Yaskawa INFORM job: X2_55B(90,0).JBI

/JOB
//NAME X2_55B(90,0)
//POS
///NPOS 393,393,393,16,0,0
///TOOL 0
///POSTYPE PULSE
///PULSE
C00000=-3448,-127156,-102318,81,81770,-493
C00001=187716,-47122,-47867,-37786,88484,55314
C00002=176173,-25216,-33637,-36582,85520,51497
C00003=173223,-25051,-31174,-36235,83113,51076
C00004=172044,-24890,-30122,-36101,82155,50902
C00005=170953,-26782,-31445,-35951,81570,50643
C00006=172044,-24890,-30122,-36101,82155,50902
C00007=171259,-26400,-31421,-35983,81846,50679
C00008=171262,-26151,-29582,-36058,81028,50950
C00009=171259,-26400,-31421,-35983,81846,50679
C00010=171893,-25290,-29924,-36099,81825,50948
C00011=170788,-22386,-27864,-35921,81544,50580
C00012=171893,-25290,-29924,-36099,81825,50948
C00013=172537,-26260,-30983,-36182,82222,51086
C00014=175513,-26532,-33522,-36519,84635,51519
C00015=174876,-38063,-42129,-21725,58370,56921
C00016=172531,-34865,-37156,-20849,56441,56328
C00017=171618,-33525,-35111,-20504,55675,56092
C00018=171621,-33203,-33229,-20744,54744,56283
C00019=171618,-33525,-35111,-20504,55675,56092
C00020=171615,-33256,-33452,-20713,54846,56260
C00021=170195,-32274,-32794,-19931,54588,55694
C00022=171615,-33256,-33452,-20713,54846,56260
C00023=172530,-34620,-35517,-21056,55613,56498
C00024=174875,-37883,-40537,-21925,57545,57094
C00025=186870,-60004,-54988,-28171,58925,61935
C00026=184052,-35224,-20919,-38155,78515,57258
C00027=176072,-20078,-10501,-37523,76109,54673
C00028=173128,-19076,-7343,-37486,73683,54259
C00029=172707,-17410,-5140,-37532,73101,54284
C00030=171611,-19099,-6383,-37450,72543,54005
C00031=172241,-18135,-5678,-37497,72864,54164
C00032=172241,-17854,-4882,-37558,72588,54263
C00033=172241,-17393,-3601,-37659,72145,54424
C00034=172241,-17647,-4307,-37604,72388,54337
C00035=171897,-14890,-2250,-37546,72359,54196
C00036=170935,-12392,-350,-37433,72036,53890
C00037=171859,-14793,-2176,-37541,72348,54182
C00038=174039,-17029,-4295,-37702,73418,54750
C00039=175523,-21167,-9806,-37619,75080,54801
C00040=174791,-34642,-26292,-23834,50951,58585
C00041=172449,-30881,-20835,-23045,48973,57976
C00042=171536,-29314,-18585,-22736,48183,57736
C00043=171539,-28594,-16381,-23083,47273,57969
C00044=171536,-29314,-18585,-22736,48183,57736
C00045=171655,-28757,-16693,-23108,47405,57991
C00046=170233,-27816,-16047,-22270,47093,57375
C00047=171655,-28757,-16693,-23108,47405,57991
C00048=172568,-30347,-18967,-23412,48199,58232
C00049=174914,-34163,-24480,-24186,50191,58839
C00050=188358,-57211,-39729,-31447,52501,64607
C00051=183618,-34426,-20428,-38127,78409,57109
C00052=176138,-20120,-10558,-37527,76149,54687
C00053=173193,-19124,-7405,-37490,73722,54273
C00054=172015,-18635,-6071,-37479,72755,54107
C00055=170924,-20442,-7388,-37397,72187,53833
C00056=172015,-18635,-6071,-37479,72755,54107
C00057=165255,-29463,-17241,-28800,66006,52931
C00058=165259,-28700,-15002,-29010,65138,53168
C00059=172949,-18171,-5639,-37573,73137,54379
C00060=171701,-15066,-3330,-37428,72734,53978
C00061=170868,-12892,-1680,-37330,72456,53714
C00062=171575,-14749,-3089,-37415,72693,53939
C00063=173186,-16870,-5921,-37451,73915,54202
C00064=175516,-21166,-9805,-37619,75076,54799
C00065=174830,-34639,-26268,-23859,50951,58604
C00066=172486,-30879,-20811,-23071,48971,57995
C00067=171574,-29313,-18562,-22761,48182,57754
C00068=171578,-28593,-16359,-23108,47271,57989
C00069=171574,-29313,-18562,-22761,48182,57754
C00070=171610,-28709,-16681,-23077,47409,57968
C00071=170190,-27766,-16033,-22239,47097,57353
C00072=171610,-28709,-16681,-23077,47409,57968
C00073=172523,-30299,-18955,-23380,48203,58209
C00074=174867,-34115,-24469,-24155,50194,58817
C00075=185275,-52966,-37377,-29840,52016,63269
C00076=182622,-32832,-19313,-38072,78076,56798
C00077=176255,-20464,-10741,-37545,76148,54738
C00078=173302,-19472,-7592,-37510,73718,54322
C00079=166116,-18702,-10817,-27686,73217,51023
C00080=166116,-18293,-9498,-27768,72681,51157
C00081=166116,-18702,-10817,-27686,73217,51023
C00082=171916,-17477,-4832,-37501,72578,54128
C00083=171280,-18444,-5544,-37452,72254,53965
C00084=171916,-17477,-4832,-37501,72578,54128
C00085=171570,-15823,-3871,-37423,72632,53954
C00086=170693,-13537,-2145,-37315,72345,53674
C00087=172061,-15821,-3938,-37462,72881,54082
C00088=175486,-21192,-9869,-37613,75083,54783
C00089=174896,-34716,-26303,-23899,50954,58635
C00090=172550,-30958,-20849,-23113,48973,58025
C00091=171637,-29393,-18600,-22803,48182,57784
C00092=171641,-28672,-16396,-23150,47273,58018
C00093=171637,-29393,-18600,-22803,48182,57784
C00094=171632,-28792,-16755,-23089,47417,57977
C00095=170210,-27851,-16107,-22251,47105,57361
C00096=171632,-28792,-16755,-23089,47417,57977
C00097=172546,-30383,-19029,-23392,48210,58218
C00098=174891,-34198,-24540,-24167,50201,58827
C00099=185175,-52762,-37248,-29786,52001,63226
C00100=183220,-33604,-19766,-38110,78246,56996
C00101=176225,-20142,-10450,-37544,76124,54733
C00102=173278,-19146,-7297,-37511,73697,54320
C00103=172099,-18657,-5963,-37501,72729,54152
C00104=171010,-20466,-7281,-37420,72160,53880
C00105=172099,-18657,-5963,-37501,72729,54152
C00106=166571,-28152,-16357,-29058,66575,53325
C00107=166571,-27514,-14492,-29226,65852,53522
C00108=172387,-18207,-5273,-37561,72696,54290
C00109=171548,-16114,-3724,-37463,72430,54020
C00110=170494,-13362,-1647,-37333,72085,53683
C00111=171073,-14893,-2806,-37405,72277,53868
C00112=172620,-14502,-2513,-37545,72964,54297
C00113=175521,-21123,-9840,-37613,75114,54788
C00114=174873,-34635,-26256,-23884,50959,58623
C00115=172529,-30877,-20800,-23097,48977,58014
C00116=171616,-29311,-18550,-22787,48188,57773
C00117=171620,-28590,-16346,-23134,47277,58007
C00118=171616,-29311,-18550,-22787,48188,57773
C00119=171603,-28722,-16701,-23071,47412,57965
C00120=170183,-27779,-16052,-22233,47100,57348
C00121=171603,-28722,-16701,-23071,47412,57965
C00122=172516,-30312,-18976,-23374,48206,58204
C00123=174861,-34128,-24489,-24150,50197,58813
C00124=179101,-45900,-49438,-15006,88631,21048
C00125=172513,-11584,-31608,-27149,87845,-38123
C00126=172121,-24857,-19443,-68057,77460,-42755
C00127=169629,-22717,-14919,-68300,75121,-42365
C00128=168643,-21776,-13037,-68423,74194,-42203
C00129=168645,-21257,-11383,-68611,73902,-41872
C00130=168643,-21776,-13037,-68423,74194,-42203
C00131=168660,-21339,-11618,-68585,73953,-41915
C00132=167619,-20808,-11231,-68547,73267,-42073
C00133=168660,-21339,-11618,-68585,73953,-41915
C00134=169647,-22299,-13520,-68449,74880,-42078
C00135=172140,-24494,-18094,-68180,77218,-42473
C00136=179100,-27267,-21132,-68321,82065,-41721
C00137=177058,-25517,-19916,-68254,80754,-42063
C00138=172070,-24843,-19439,-68055,77427,-42764
C00139=169578,-22699,-14913,-68297,75090,-42374
C00140=168592,-21759,-13031,-68421,74162,-42212
C00141=168594,-21241,-11375,-68608,73870,-41880
C00142=168592,-21759,-13031,-68421,74162,-42212
C00143=168700,-21363,-11631,-68587,73978,-41908
C00144=167658,-20834,-11246,-68549,73291,-42065
C00145=168700,-21363,-11631,-68587,73978,-41908
C00146=169687,-22325,-13534,-68451,74905,-42070
C00147=172181,-24516,-18104,-68183,77243,-42465
C00148=177058,-25517,-19916,-68254,80754,-42063
C00149=178325,-24532,-19230,-68277,81638,-41928
C00150=172107,-24845,-19446,-68056,77454,-42760
C00151=169616,-22704,-14920,-68297,75115,-42370
C00152=168630,-22174,-14386,-68271,74432,-42481
C00153=168630,-21922,-13548,-68363,74279,-42313
C00154=168630,-22174,-14386,-68271,74432,-42481
C00155=167254,-20761,-13369,-68184,73550,-42717
C00156=168630,-22174,-14386,-68271,74432,-42481
C00157=169618,-22273,-13490,-68449,74858,-42080
C00158=172110,-24469,-18066,-68180,77195,-42476
C00159=178325,-24532,-19230,-68277,81638,-41928
C00160=176815,-23437,-18422,-68227,80649,-42160
C00161=172146,-24955,-19493,-68063,77470,-42744
C00162=169652,-22814,-14970,-68305,75130,-42353
C00163=168665,-21875,-13087,-68429,74203,-42192
C00164=168667,-21355,-11432,-68616,73909,-41860
C00165=168665,-21875,-13087,-68429,74203,-42192
C00166=168662,-21419,-11696,-68583,73957,-41918
C00167=167620,-20888,-11311,-68545,73271,-42076
C00168=168662,-21419,-11696,-68583,73957,-41918
C00169=169650,-22379,-13598,-68447,74884,-42081
C00170=172143,-24573,-18170,-68179,77222,-42475
C00171=176815,-23437,-18422,-68227,80649,-42160
C00172=177723,-27338,-20753,-73480,80899,-41496
C00173=173318,-27034,-20539,-73385,77850,-41980
C00174=170566,-24945,-16343,-73635,75471,-41597
C00175=168745,-21940,-12752,-73770,74001,-41488
C00176=168745,-21543,-11513,-73914,73830,-41233
C00177=168745,-21940,-12752,-73770,74001,-41488
C00178=167687,-21056,-12116,-73735,73288,-41631
C00179=168745,-21940,-12752,-73770,74001,-41488
C00180=170579,-24581,-15077,-73772,75297,-41328
C00181=173331,-26714,-19314,-73495,77675,-41714
C00182=177723,-27338,-20753,-73480,80899,-41496
C00183=178463,-3707,1935,-68390,87302,-39636
C00184=172445,-1687,3602,-68547,83267,-40440
C00185=171155,2365,8138,-68637,82124,-40308
C00186=169346,2928,9772,-68759,80632,-40240
C00187=168978,-317,7268,-68782,80335,-40236
C00188=168639,-4450,3875,-68796,80092,-40264
C00189=168178,-8509,681,-68823,79735,-40271
C00190=167808,-11173,-1351,-68851,79442,-40266
C00191=167512,-13424,-3126,-68866,79215,-40276
C00192=170518,-14544,-5815,-68770,81540,-41125
C00193=171276,-16033,-7526,-68427,80959,-50953
C00194=176138,-7665,-1065,-68313,84347,-50442
C00195=175728,4349,8139,-68463,85593,-40138
C00196=172451,-1962,2819,-68519,83404,-40586
C00197=170217,-243,7278,-68749,81179,-40082
C00198=168682,3850,12028,-68899,79836,-39929
C00199=168320,-294,8663,-68919,79564,-39952
C00200=167945,-5454,4438,-68970,78444,-40143
C00201=167170,-12539,-831,-69280,75932,-44117
C00202=166914,-13716,-1698,-69168,76543,-48053
C00203=168751,-15418,-4687,-68668,78708,-50672
C00204=171281,-16312,-8291,-68386,81093,-51093
C00205=176223,-7788,-1720,-68290,84540,-50575
C00206=175841,4947,9210,-68476,85532,-39971
C00207=172439,-1632,3648,-68547,83263,-40441
C00208=170207,122,8144,-68792,81039,-39934
C00209=169582,3762,12383,-68907,80337,-39699
C00210=169205,-1273,8190,-68921,80079,-39742
C00211=168949,-4829,5248,-68968,79052,-39936
C00212=168747,-7437,3182,-69019,78039,-40097
C00213=168400,-11411,49,-69099,75859,-40464
C00214=168049,-14366,-2154,-69161,74008,-40742
C00215=167878,-15531,-2988,-69182,74134,-40673
C00216=167909,-10329,250,-68068,79474,-40087
C00217=167962,-8065,2008,-67933,82039,-39608
C00218=168741,-15055,-3851,-68723,78573,-50532
C00219=171270,-15979,-7485,-68426,80956,-50955
C00220=176912,-6106,181,-68292,84880,-50353
C00221=175080,3284,7783,-68495,85030,-40084
C00222=172448,-1714,3579,-68547,83270,-40439
C00223=170215,38,8073,-68791,81044,-39933
C00224=169530,3059,11777,-68909,80304,-39708
C00225=169167,-1208,8273,-68926,80049,-39741
C00226=168895,-5244,4985,-68982,78994,-39919
C00227=168721,-7713,2972,-69022,78019,-40095
C00228=168321,-11533,70,-69119,75776,-40439
C00229=168019,-14335,-2124,-69163,73986,-40743
C00230=167869,-15557,-2996,-69185,74125,-40670
C00231=167778,-15678,-3083,-69135,76109,-40273
C00232=168308,-1085,8366,-68428,86286,-38506
C00233=168749,-15137,-3913,-68724,78577,-50529
C00234=171279,-16061,-7546,-68427,80961,-50952
C00235=176975,-6087,196,-68290,84923,-50345
C00236=175436,4075,8459,-68486,85264,-40032
C00237=172442,-1659,3624,-68547,83265,-40441
C00238=170209,94,8121,-68791,81041,-39934
C00239=169521,3688,12369,-68916,80282,-39689
C00240=169178,-1205,8258,-68923,80058,-39744
C00241=168951,-4837,5280,-68974,79043,-39923
C00242=168871,-5612,4655,-68979,78986,-39928
C00243=168324,-12009,-390,-69107,75794,-40458
C00244=167899,-15618,-3071,-69178,74154,-40675
C00245=168117,-12377,-741,-68965,78498,-39952
C00246=168316,-5643,4501,-68586,83486,-39095
C00247=169562,-13065,-2936,-68632,79303,-50620
C00248=171273,-16006,-7506,-68427,80957,-50954
C00249=176232,-7453,-896,-68311,84412,-50431
C00250=176110,15147,-7571,-16904,97824,-889
C00251=169929,-46392,-55011,-1489,81060,44357
C00252=178847,-41200,-24878,-45467,45731,82659
C00253=176214,-37608,-19575,-45318,43383,82417
C00254=175671,-33630,-15830,-45260,42922,82348
C00255=175825,-32530,-15066,-45264,43068,82357
C00256=178049,-27664,-11799,-47846,47063,84437
C00257=178346,-25405,-10245,-47840,47361,84442
C00258=178686,-23359,-8771,-47863,47635,84481
C00259=179298,-27755,-13076,-47829,48231,84493
C00260=181844,-30788,-18177,-47745,50662,84564
C00261=174365,-16035,-7463,-23225,65722,49139
C00262=172039,-13164,-2259,-22946,63476,48682
C00263=170681,-8939,2085,-22689,62636,48310
C00264=168716,-14063,-1663,-20852,60530,45982
C00265=168210,-15866,-3076,-20705,60349,45807
C00266=167705,-17394,-4214,-20570,60144,45641
C00267=168908,-9574,565,-22819,69097,42788
C00268=170886,-12368,-2848,-23069,70258,43317
C00269=173248,-14965,-7813,-23249,72509,43767
C00270=172938,-13150,-5784,-34661,81894,69122
C00271=170592,-13671,-3251,-34736,79423,68935
C00272=169013,-12050,-743,-34751,78192,68673
C00273=168391,-10413,528,-34716,77985,68483
C00274=167212,-7347,2971,-34654,77563,68126
C00275=167368,-11109,1537,-37136,72671,67957
C00276=169061,-13362,-1350,-37170,73898,68258
C00277=171567,-13522,-4340,-37101,76395,68464
C00278=179365,-30795,-16721,-37645,78767,70970
C00279=189901,-62154,-47134,-47848,53538,74187
C00280=178827,-45311,-37716,-41873,49979,80234
C00281=176196,-42115,-32789,-41416,47672,79900
C00282=175621,-38539,-29280,-41324,47154,79828
C00283=175830,-37491,-28575,-41455,47414,79922
C00284=176568,-36338,-27837,-42536,48701,80694
C00285=177913,-33249,-25871,-44214,51091,81919
C00286=178266,-30726,-24137,-44250,51432,81940
C00287=178622,-27514,-21859,-44263,51790,81950
C00288=179281,-31896,-26227,-44296,52442,81981
C00289=181826,-34468,-30902,-44523,54848,82142
C00290=174316,-20812,-35323,-21564,79352,46486
C00291=171992,-19198,-31213,-21065,77169,46035
C00292=171153,-17227,-28586,-20882,76391,45864
C00293=169593,-21753,-31892,-19124,74559,43851
C00294=168812,-24435,-33772,-18910,74171,43627
C00295=168062,-26842,-35420,-18710,73789,43414
C00296=169770,-16807,-29422,-21714,83022,40480
C00297=169547,-17498,-29909,-21673,82913,40417
C00298=170841,-17822,-31354,-21899,83925,40699
C00299=173201,-19163,-35240,-22305,86132,41137
C00300=172907,-17608,-30546,-34532,92651,65775
C00301=170563,-19319,-28972,-34275,90177,65595
C00302=169577,-19876,-27906,-34181,88999,65557
C00303=168529,-16782,-25766,-34081,88801,65197
C00304=167923,-15565,-24727,-34164,88196,64970
C00305=167964,-19498,-26291,-35768,83354,64607
C00306=169032,-19661,-27621,-35877,84402,64708
C00307=171538,-18685,-29668,-36163,86886,64924
C00308=178275,-34785,-40895,-36932,88626,67129
C00309=191077,-58387,-34695,-51576,50395,82052
C00310=178834,-41148,-24847,-45459,45731,82652
C00311=176205,-37556,-19542,-45310,43382,82411
C00312=175763,-33644,-15876,-45294,42982,82374
C00313=178032,-28543,-12452,-47893,47019,84460
C00314=178404,-25994,-10760,-47830,47404,84453
C00315=178792,-23615,-9141,-47838,47760,84471
C00316=179288,-27703,-13041,-47822,48229,84487
C00317=181832,-30737,-18143,-47737,50660,84558
C00318=174357,-15982,-7423,-23222,65723,49136
C00319=172031,-13111,-2218,-22944,63477,48679
C00320=170520,-8947,1823,-22613,62739,48224
C00321=170034,-11263,-69,-22486,62583,48061
C00322=169470,-13204,-1541,-22355,62344,47883
C00323=168361,-16702,-4145,-22089,61865,47531
C00324=168865,-9474,239,-22775,69314,42731
C00325=170879,-12314,-2806,-23068,70257,43314
C00326=173241,-14911,-7773,-23247,72510,43764
C00327=172940,-13092,-5769,-34660,81912,69117
C00328=170596,-13616,-3238,-34734,79442,68930
C00329=168939,-11997,-1091,-34723,78363,68588
C00330=168389,-10110,342,-34686,78206,68407
C00331=167070,-6484,3213,-34619,77749,68010
C00332=167299,-10933,1331,-37095,72823,67875
C00333=169065,-13308,-1339,-37166,73916,68253
C00334=171571,-13466,-4327,-37098,76413,68459
C00335=178312,-28732,-15356,-37588,78485,70620
C00336=191277,-58648,-34832,-51660,50475,82922
C00337=178852,-41226,-24894,-45472,45733,82663
C00338=176220,-37634,-19591,-45323,43383,82420
C00339=175685,-33946,-16007,-45315,42889,82377
C00340=175835,-32522,-15044,-45277,43065,82364
C00341=178144,-27733,-11903,-47880,47136,84457
C00342=178393,-25451,-10265,-47844,47377,84457
C00343=178672,-23784,-9159,-47826,47648,84464
C00344=179304,-27780,-13094,-47832,48232,84495
C00345=181850,-30813,-18194,-47748,50663,84567
C00346=174368,-16065,-7493,-23225,65726,49140
C00347=172043,-13195,-2289,-22946,63480,48682
C00348=171164,-7550,3016,-22790,62898,48455
C00349=170866,-8989,1826,-22712,62814,48348
C00350=170143,-11437,8,-22546,62486,48122
C00351=169193,-14739,-2522,-22318,62099,47819
C00352=169244,-9393,584,-22743,68342,43554
C00353=170889,-12399,-2879,-23069,70262,43318
C00354=173252,-14995,-7844,-23249,72513,43768
C00355=172951,-13173,-5831,-34660,81913,69121
C00356=170605,-13697,-3300,-34735,79444,68934
C00357=169521,-10404,420,-34756,78511,68787
C00358=168984,-8925,1564,-34730,78334,68616
C00359=167678,-5351,4395,-34667,77878,68219
C00360=170004,-9650,4792,-41331,72244,71659
C00361=169881,-12181,-477,-37221,74307,68468
C00362=171580,-13547,-4389,-37099,76414,68462
C00363=179014,-30130,-16303,-37625,78683,70850
C00364=192370,-59799,-35433,-52082,50945,77766
C00365=178840,-41174,-24863,-45463,45731,82656
C00366=176209,-37582,-19559,-45314,43383,82414
C00367=175858,-33709,-16041,-45280,43083,82373
C00368=175847,-33097,-15509,-45291,43063,82377
C00369=178181,-27613,-11893,-47837,47190,84441
C00370=178483,-25011,-10021,-47840,47478,84452
C00371=178690,-24031,-9393,-47845,47668,84462
C00372=179293,-27729,-13059,-47826,48231,84490
C00373=181839,-30763,-18160,-47741,50661,84561
C00374=174361,-16008,-7442,-23223,65722,49137
C00375=172034,-13138,-2238,-22945,63477,48680
C00376=171207,-7845,2636,-22781,62991,48446
C00377=170272,-11167,86,-22561,62606,48149
C00378=169822,-12966,-1346,-22450,62442,48001
C00379=168964,-15587,-3284,-22246,62068,47732
C00380=173943,-1511,8904,-29878,72865,47458
C00381=172046,-12965,-4840,-23146,71432,43525
C00382=173245,-14938,-7793,-23248,72510,43766
C00383=172944,-13119,-5789,-34660,81912,69118
C00384=170599,-13643,-3259,-34734,79442,68931
C00385=169526,-10552,102,-34744,78615,68757
C00386=169161,-9437,984,-34729,78491,68643
C00387=167403,-4604,4769,-34640,77906,68103
C00388=171806,-13548,4066,-45686,69255,74076
C00389=169068,-13335,-1360,-37167,73916,68254
C00390=171574,-13493,-4347,-37099,76413,68460
C00391=179991,-31915,-17499,-37671,78963,71169
C00392=-3448,-127156,-102318,81,81770,-493
BC00000=88064,523889,1075193
BC00001=92522,523889,1075139
BC00002=92522,523889,1075139
BC00003=92522,523889,1075139
BC00004=92522,523889,1075139
BC00005=92522,523889,1075139
BC00006=92522,523889,1075139
BC00007=92522,523889,1075139
BC00008=92522,523889,1075139
BC00009=92522,523889,1075139
BC00010=92522,523889,1075139
BC00011=92522,523889,1075139
BC00012=92522,523889,1075139
BC00013=92522,523889,1075139
BC00014=92522,523889,1075139
BC00015=117731,523889,1075139
BC00016=117731,523889,1075139
BC00017=117731,523889,1075139
BC00018=117731,523889,1075139
BC00019=117731,523889,1075139
BC00020=117731,523889,1075139
BC00021=117731,523889,1075139
BC00022=117731,523889,1075139
BC00023=117731,523889,1075139
BC00024=117731,523889,1075139
BC00025=117731,523889,1075139
BC00026=92535,523889,1039496
BC00027=92535,523889,1039496
BC00028=92535,523889,1039496
BC00029=92535,523889,1039496
BC00030=92535,523889,1039496
BC00031=92535,523889,1039496
BC00032=92535,523889,1039496
BC00033=92535,523889,1039496
BC00034=92535,523889,1039496
BC00035=92535,523889,1039496
BC00036=92535,523889,1039496
BC00037=92535,523889,1039496
BC00038=92535,523889,1039496
BC00039=92535,523889,1039496
BC00040=117708,523889,1001261
BC00041=117708,523889,1001261
BC00042=117708,523889,1001261
BC00043=117708,523889,1001261
BC00044=117708,523889,1001261
BC00045=117708,523889,1001261
BC00046=117708,523889,1001261
BC00047=117708,523889,1001261
BC00048=117708,523889,1001261
BC00049=117708,523889,1001261
BC00050=117708,523889,1001261
BC00051=92605,523889,877547
BC00052=92605,523889,877547
BC00053=92605,523889,877547
BC00054=92605,523889,877547
BC00055=92605,523889,877547
BC00056=92605,523889,877547
BC00057=92605,523889,877547
BC00058=92605,523889,877547
BC00059=92605,523889,877547
BC00060=92605,523889,877547
BC00061=92605,523889,877547
BC00062=92605,523889,877547
BC00063=92605,523889,877547
BC00064=92605,523889,877547
BC00065=117541,523889,839285
BC00066=117541,523889,839285
BC00067=117541,523889,839285
BC00068=117541,523889,839285
BC00069=117541,523889,839285
BC00070=117541,523889,839285
BC00071=117541,523889,839285
BC00072=117541,523889,839285
BC00073=117541,523889,839285
BC00074=117541,523889,839285
BC00075=117541,523889,839285
BC00076=92484,523889,715304
BC00077=92484,523889,715304
BC00078=92484,523889,715304
BC00079=92484,523889,715304
BC00080=92484,523889,715304
BC00081=92484,523889,715304
BC00082=92484,523889,715304
BC00083=92484,523889,715304
BC00084=92484,523889,715304
BC00085=92484,523889,715304
BC00086=92484,523889,715304
BC00087=92484,523889,715304
BC00088=92484,523889,715304
BC00089=117712,523889,677277
BC00090=117712,523889,677277
BC00091=117712,523889,677277
BC00092=117712,523889,677277
BC00093=117712,523889,677277
BC00094=117712,523889,677277
BC00095=117712,523889,677277
BC00096=117712,523889,677277
BC00097=117712,523889,677277
BC00098=117712,523889,677277
BC00099=117712,523889,677277
BC00100=92665,523889,553782
BC00101=92665,523889,553782
BC00102=92665,523889,553782
BC00103=92665,523889,553782
BC00104=92665,523889,553782
BC00105=92665,523889,553782
BC00106=92665,523889,553782
BC00107=92665,523889,553782
BC00108=92665,523889,553782
BC00109=92665,523889,553782
BC00110=92665,523889,553782
BC00111=92665,523889,553782
BC00112=92665,523889,553782
BC00113=92665,523889,553782
BC00114=117593,523889,515943
BC00115=117593,523889,515943
BC00116=117593,523889,515943
BC00117=117593,523889,515943
BC00118=117593,523889,515943
BC00119=117593,523889,515943
BC00120=117593,523889,515943
BC00121=117593,523889,515943
BC00122=117593,523889,515943
BC00123=117593,523889,515943
BC00124=88297,523889,479689
BC00125=36680,523889,415813
BC00126=28310,523889,405455
BC00127=28310,523889,405455
BC00128=29106,522353,405455
BC00129=29106,522353,405455
BC00130=29106,522353,405455
BC00131=29106,522353,405455
BC00132=29106,522353,405455
BC00133=29106,522353,405455
BC00134=29106,522353,405455
BC00135=29106,522353,405455
BC00136=29106,522353,405455
BC00137=29225,522353,566726
BC00138=29225,522353,566726
BC00139=29225,522353,566726
BC00140=29225,522353,566726
BC00141=29225,522353,566726
BC00142=29225,522353,566726
BC00143=29225,522353,566726
BC00144=29225,522353,566726
BC00145=29225,522353,566726
BC00146=29225,522353,566726
BC00147=29225,522353,566726
BC00148=29225,522353,566726
BC00149=28944,522353,728798
BC00150=28944,522353,728798
BC00151=28944,522353,728798
BC00152=28944,522353,728798
BC00153=28944,522353,728798
BC00154=28944,522353,728798
BC00155=28944,522353,728798
BC00156=28944,522353,728798
BC00157=28944,522353,728798
BC00158=28944,522353,728798
BC00159=28944,522353,728798
BC00160=29066,522353,891103
BC00161=29066,522353,891103
BC00162=29066,522353,891103
BC00163=29066,522353,891103
BC00164=29066,522353,891103
BC00165=29066,522353,891103
BC00166=29066,522353,891103
BC00167=29066,522353,891103
BC00168=29066,522353,891103
BC00169=29066,522353,891103
BC00170=29066,522353,891103
BC00171=29066,522353,891103
BC00172=26330,522353,1022235
BC00173=26330,522353,1022235
BC00174=26330,522353,1022235
BC00175=26330,522353,1022235
BC00176=26330,522353,1022235
BC00177=26330,522353,1022235
BC00178=26330,522353,1022235
BC00179=26330,522353,1022235
BC00180=26330,522353,1022235
BC00181=26330,522353,1022235
BC00182=26330,522353,1022235
BC00183=28832,522353,754426
BC00184=28036,523889,754426
BC00185=28036,523889,754426
BC00186=28832,522353,754426
BC00187=28832,522353,754426
BC00188=28832,522353,754426
BC00189=28832,522353,754426
BC00190=28832,522353,754426
BC00191=28832,522353,754426
BC00192=28832,522353,754426
BC00193=28832,522353,754426
BC00194=28832,522353,754426
BC00195=28825,522353,1075139
BC00196=28825,522353,1075139
BC00197=28825,522353,1075139
BC00198=28825,522353,1075139
BC00199=28825,522353,1075139
BC00200=28825,522353,1075139
BC00201=28825,522353,1075139
BC00202=28825,522353,1075139
BC00203=28825,522353,1075139
BC00204=28825,522353,1075139
BC00205=28825,522353,1075139
BC00206=28839,522353,431016
BC00207=28839,522353,431016
BC00208=28839,522353,431016
BC00209=28839,522353,431016
BC00210=28839,522353,431016
BC00211=28839,522353,431016
BC00212=28839,522353,431016
BC00213=28839,522353,431016
BC00214=28839,522353,431016
BC00215=28839,522353,431016
BC00216=28839,522353,431016
BC00217=28839,522353,431016
BC00218=28839,522353,431016
BC00219=28839,522353,431016
BC00220=28839,522353,431016
BC00221=28829,522353,916535
BC00222=28829,522353,916535
BC00223=28829,522353,916535
BC00224=28829,522353,916535
BC00225=28829,522353,916535
BC00226=28829,522353,916535
BC00227=28829,522353,916535
BC00228=28829,522353,916535
BC00229=28829,522353,916535
BC00230=28829,522353,916535
BC00231=28829,522353,916535
BC00232=28829,522353,916535
BC00233=28829,522353,916535
BC00234=28829,522353,916535
BC00235=28829,522353,916535
BC00236=28835,522353,592318
BC00237=28835,522353,592318
BC00238=28835,522353,592318
BC00239=28835,522353,592318
BC00240=28835,522353,592318
BC00241=28835,522353,592318
BC00242=28835,522353,592318
BC00243=28835,522353,592318
BC00244=28835,522353,592318
BC00245=28835,522352,592316
BC00246=28835,522352,592316
BC00247=28835,522353,592318
BC00248=28835,522353,592318
BC00249=28835,522353,592318
BC00250=67844,522353,695135
BC00251=94775,523889,768216
BC00252=112941,523889,816097
BC00253=112941,523889,816097
BC00254=112941,523889,816097
BC00255=112941,523889,816097
BC00256=112941,523889,816097
BC00257=112941,523889,816097
BC00258=112941,523889,816097
BC00259=112941,523889,816097
BC00260=112941,523889,816097
BC00261=118115,523889,907170
BC00262=118115,523889,907170
BC00263=118115,523889,907170
BC00264=118115,523889,907170
BC00265=118115,523889,907170
BC00266=118115,523889,907170
BC00267=118115,523889,907170
BC00268=118115,523889,907170
BC00269=118115,523889,907170
BC00270=88032,523889,888291
BC00271=88032,523889,888291
BC00272=88032,523889,888291
BC00273=88032,523889,888291
BC00274=88032,523889,888291
BC00275=88032,523889,888291
BC00276=88032,523889,888291
BC00277=88032,523889,888291
BC00278=88032,523889,888291
BC00279=112934,523889,1075139
BC00280=112934,523889,1075139
BC00281=112934,523889,1075139
BC00282=112934,523889,1075139
BC00283=112934,523889,1075139
BC00284=112934,523889,1075139
BC00285=112934,523889,1075139
BC00286=112934,523889,1075139
BC00287=112934,523889,1075139
BC00288=112934,523889,1075139
BC00289=112934,523889,1075139
BC00290=118108,523889,1075139
BC00291=118108,523889,1075139
BC00292=118108,523889,1075139
BC00293=118108,523889,1075139
BC00294=118108,523889,1075139
BC00295=118108,523889,1075139
BC00296=118108,523889,1075139
BC00297=118108,523889,1075139
BC00298=118108,523889,1075139
BC00299=118108,523889,1075139
BC00300=88054,523889,1075139
BC00301=88054,523889,1075139
BC00302=88054,523888,1075137
BC00303=88054,523889,1075139
BC00304=88054,523889,1075139
BC00305=88054,523889,1075139
BC00306=88054,523889,1075139
BC00307=88054,523889,1075139
BC00308=88054,523889,1075139
BC00309=112948,523889,492686
BC00310=112948,523889,492686
BC00311=112948,523889,492686
BC00312=112948,523889,492686
BC00313=112948,523889,492686
BC00314=112948,523889,492686
BC00315=112948,523889,492686
BC00316=112948,523889,492686
BC00317=112948,523889,492686
BC00318=118122,523889,583760
BC00319=118122,523889,583760
BC00320=118122,523889,583760
BC00321=118122,523889,583760
BC00322=118122,523889,583760
BC00323=118122,523889,583760
BC00324=118122,523889,583760
BC00325=118122,523889,583760
BC00326=118122,523889,583760
BC00327=88067,523889,564693
BC00328=88067,523889,564693
BC00329=88067,523889,564693
BC00330=88067,523889,564693
BC00331=88067,523889,564693
BC00332=88067,523889,564693
BC00333=88067,523889,564693
BC00334=88067,523889,564693
BC00335=88067,523889,564693
BC00336=112938,523889,978206
BC00337=112938,523889,978206
BC00338=112938,523889,978206
BC00339=112938,523889,978206
BC00340=112938,523889,978206
BC00341=112938,523889,978206
BC00342=112938,523889,978206
BC00343=112938,523889,978206
BC00344=112938,523889,978206
BC00345=112938,523889,978206
BC00346=118112,523889,1069230
BC00347=118112,523889,1069230
BC00348=118112,523889,1069230
BC00349=118112,523889,1069230
BC00350=118112,523889,1069230
BC00351=118112,523889,1069230
BC00352=118111,523889,1069227
BC00353=118112,523889,1069230
BC00354=118112,523889,1069230
BC00355=88057,523889,1050213
BC00356=88057,523889,1050213
BC00357=88057,523889,1050213
BC00358=88057,523889,1050213
BC00359=88057,523889,1050213
BC00360=88057,523889,1050213
BC00361=88057,523889,1050213
BC00362=88057,523889,1050213
BC00363=88057,523889,1050213
BC00364=112944,523889,653988
BC00365=112944,523889,653988
BC00366=112944,523889,653988
BC00367=112944,523889,653988
BC00368=112944,523889,653988
BC00369=112944,523889,653988
BC00370=112944,523889,653988
BC00371=112944,523889,653988
BC00372=112944,523889,653988
BC00373=112944,523889,653988
BC00374=118118,523889,745062
BC00375=118118,523889,745062
BC00376=118118,523889,745062
BC00377=118118,523889,745062
BC00378=118118,523889,745062
BC00379=118118,523889,745062
BC00380=118118,523889,745062
BC00381=118118,523889,745062
BC00382=118118,523889,745062
BC00383=88064,523889,725995
BC00384=88064,523889,725995
BC00385=88064,523889,725995
BC00386=88064,523889,725995
BC00387=88064,523889,725995
BC00388=88064,523889,725995
BC00389=88064,523889,725995
BC00390=88064,523889,725995
BC00391=88064,555625,725995
BC00392=88064,523889,1075193
EC00000=-798156,-183832
EC00001=-798156,-183832
EC00002=-798156,-183832
EC00003=-798156,-183832
EC00004=-798156,-183832
EC00005=-798156,-183832
EC00006=-798156,-183832
EC00007=-798156,-183832
EC00008=-798156,-183832
EC00009=-798156,-183832
EC00010=-798156,-183832
EC00011=-798156,-183832
EC00012=-798156,-183832
EC00013=-798156,-183832
EC00014=-798156,-183832
EC00015=-798156,-183832
EC00016=-798156,-183832
EC00017=-798156,-183832
EC00018=-798156,-183832
EC00019=-798156,-183832
EC00020=-798156,-183832
EC00021=-798156,-183832
EC00022=-798156,-183832
EC00023=-798156,-183832
EC00024=-798156,-183832
EC00025=-798156,-183832
EC00026=-798156,-183832
EC00027=-798156,-183832
EC00028=-798156,-183832
EC00029=-798156,-183832
EC00030=-798156,-183832
EC00031=-798156,-183832
EC00032=-798156,-183832
EC00033=-798156,-183832
EC00034=-798156,-183832
EC00035=-798156,-183832
EC00036=-798156,-183832
EC00037=-798156,-183832
EC00038=-798156,-183832
EC00039=-798156,-183832
EC00040=-798156,-183832
EC00041=-798156,-183832
EC00042=-798156,-183832
EC00043=-798156,-183832
EC00044=-798156,-183832
EC00045=-798156,-183832
EC00046=-798156,-183832
EC00047=-798156,-183832
EC00048=-798156,-183832
EC00049=-798156,-183832
EC00050=-798156,-183832
EC00051=-798156,-183832
EC00052=-798156,-183832
EC00053=-798156,-183832
EC00054=-798156,-183832
EC00055=-798156,-183832
EC00056=-798156,-183832
EC00057=-798156,-183832
EC00058=-798156,-183832
EC00059=-798156,-183832
EC00060=-798156,-183832
EC00061=-798156,-183832
EC00062=-798156,-183832
EC00063=-798156,-183832
EC00064=-798156,-183832
EC00065=-798156,-183832
EC00066=-798156,-183832
EC00067=-798156,-183832
EC00068=-798156,-183832
EC00069=-798156,-183832
EC00070=-798156,-183832
EC00071=-798156,-183832
EC00072=-798156,-183832
EC00073=-798156,-183832
EC00074=-798156,-183832
EC00075=-798156,-183832
EC00076=-798156,-183832
EC00077=-798156,-183832
EC00078=-798156,-183832
EC00079=-798156,-183832
EC00080=-798156,-183832
EC00081=-798156,-183832
EC00082=-798156,-183832
EC00083=-798156,-183832
EC00084=-798156,-183832
EC00085=-798156,-183832
EC00086=-798156,-183832
EC00087=-798156,-183832
EC00088=-798156,-183832
EC00089=-798156,-183832
EC00090=-798156,-183832
EC00091=-798156,-183832
EC00092=-798156,-183832
EC00093=-798156,-183832
EC00094=-798156,-183832
EC00095=-798156,-183832
EC00096=-798156,-183832
EC00097=-798156,-183832
EC00098=-798156,-183832
EC00099=-798156,-183832
EC00100=-798156,-183832
EC00101=-798156,-183832
EC00102=-798156,-183832
EC00103=-798156,-183832
EC00104=-798156,-183832
EC00105=-798156,-183832
EC00106=-798156,-183832
EC00107=-798156,-183832
EC00108=-798156,-183832
EC00109=-798156,-183832
EC00110=-798156,-183832
EC00111=-798156,-183832
EC00112=-798156,-183832
EC00113=-798156,-183832
EC00114=-798156,-183832
EC00115=-798156,-183832
EC00116=-798156,-183832
EC00117=-798156,-183832
EC00118=-798156,-183832
EC00119=-798156,-183832
EC00120=-798156,-183832
EC00121=-798156,-183832
EC00122=-798156,-183832
EC00123=-798156,-183832
EC00124=-798156,-183832
EC00125=-798156,-183832
EC00126=-798156,-183832
EC00127=-798156,-183832
EC00128=-798156,-183832
EC00129=-798156,-183832
EC00130=-798156,-183832
EC00131=-798156,-183832
EC00132=-798156,-183832
EC00133=-798156,-183832
EC00134=-798156,-183832
EC00135=-798156,-183832
EC00136=-798156,-183832
EC00137=-798156,-183832
EC00138=-798156,-183832
EC00139=-798156,-183832
EC00140=-798156,-183832
EC00141=-798156,-183832
EC00142=-798156,-183832
EC00143=-798156,-183832
EC00144=-798156,-183832
EC00145=-798156,-183832
EC00146=-798156,-183832
EC00147=-798156,-183832
EC00148=-798156,-183832
EC00149=-798156,-183832
EC00150=-798156,-183832
EC00151=-798156,-183832
EC00152=-798156,-183832
EC00153=-798156,-183832
EC00154=-798156,-183832
EC00155=-798156,-183832
EC00156=-798156,-183832
EC00157=-798156,-183832
EC00158=-798156,-183832
EC00159=-798156,-183832
EC00160=-798156,-183832
EC00161=-798156,-183832
EC00162=-798156,-183832
EC00163=-798156,-183832
EC00164=-798156,-183832
EC00165=-798156,-183832
EC00166=-798156,-183832
EC00167=-798156,-183832
EC00168=-798156,-183832
EC00169=-798156,-183832
EC00170=-798156,-183832
EC00171=-798156,-183832
EC00172=-798156,-183832
EC00173=-798156,-183832
EC00174=-798156,-183832
EC00175=-798156,-183832
EC00176=-798156,-183832
EC00177=-798156,-183832
EC00178=-798156,-183832
EC00179=-798156,-183832
EC00180=-798156,-183832
EC00181=-798156,-183832
EC00182=-798156,-183832
EC00183=-798156,-183832
EC00184=-798156,-183832
EC00185=-798156,-183832
EC00186=-798156,-183832
EC00187=-798156,-183832
EC00188=-798156,-183832
EC00189=-798156,-183832
EC00190=-798156,-183832
EC00191=-798156,-183832
EC00192=-798156,-183832
EC00193=-798156,-183832
EC00194=-798156,-183832
EC00195=-798156,-183832
EC00196=-798156,-183832
EC00197=-798156,-183832
EC00198=-798156,-183832
EC00199=-798156,-183832
EC00200=-798156,-183832
EC00201=-798156,-183832
EC00202=-798156,-183832
EC00203=-798156,-183832
EC00204=-798156,-183832
EC00205=-798156,-183832
EC00206=-798156,-183832
EC00207=-798156,-183832
EC00208=-798156,-183832
EC00209=-798156,-183832
EC00210=-798156,-183832
EC00211=-798156,-183832
EC00212=-798156,-183832
EC00213=-798156,-183832
EC00214=-798156,-183832
EC00215=-798156,-183832
EC00216=-798156,-183832
EC00217=-798156,-183832
EC00218=-798156,-183832
EC00219=-798156,-183832
EC00220=-798156,-183832
EC00221=-798156,-183832
EC00222=-798156,-183832
EC00223=-798156,-183832
EC00224=-798156,-183832
EC00225=-798156,-183832
EC00226=-798156,-183832
EC00227=-798156,-183832
EC00228=-798156,-183832
EC00229=-798156,-183832
EC00230=-798156,-183832
EC00231=-798156,-183832
EC00232=-798156,-183832
EC00233=-798156,-183832
EC00234=-798156,-183832
EC00235=-798156,-183832
EC00236=-798156,-183832
EC00237=-798156,-183832
EC00238=-798156,-183832
EC00239=-798156,-183832
EC00240=-798156,-183832
EC00241=-798156,-183832
EC00242=-798156,-183832
EC00243=-798156,-183832
EC00244=-798156,-183832
EC00245=-798155,-183832
EC00246=-798155,-183832
EC00247=-798156,-183832
EC00248=-798156,-183832
EC00249=-798156,-183832
EC00250=-798156,-183832
EC00251=-798156,-183832
EC00252=-798156,-183832
EC00253=-798156,-183832
EC00254=-798156,-183832
EC00255=-798156,-183832
EC00256=-798156,-183832
EC00257=-798156,-183832
EC00258=-798156,-183832
EC00259=-798156,-183832
EC00260=-798156,-183832
EC00261=-798156,-183832
EC00262=-798156,-183832
EC00263=-798156,-183832
EC00264=-798156,-183832
EC00265=-798156,-183832
EC00266=-798156,-183832
EC00267=-798156,-183832
EC00268=-798156,-183832
EC00269=-798156,-183832
EC00270=-798156,-183832
EC00271=-798156,-183832
EC00272=-798156,-183832
EC00273=-798156,-183832
EC00274=-798156,-183832
EC00275=-798156,-183832
EC00276=-798156,-183832
EC00277=-798156,-183832
EC00278=-798156,-183832
EC00279=-798156,-183832
EC00280=-798156,-183832
EC00281=-798156,-183832
EC00282=-798156,-183832
EC00283=-798156,-183832
EC00284=-798156,-183832
EC00285=-798156,-183832
EC00286=-798156,-183832
EC00287=-798156,-183832
EC00288=-798156,-183832
EC00289=-798156,-183832
EC00290=-798156,-183832
EC00291=-798156,-183832
EC00292=-798156,-183832
EC00293=-798156,-183832
EC00294=-798156,-183832
EC00295=-798156,-183832
EC00296=-798156,-183832
EC00297=-798156,-183832
EC00298=-798156,-183832
EC00299=-798156,-183832
EC00300=-798156,-183832
EC00301=-798156,-183832
EC00302=-798155,-183833
EC00303=-798156,-183832
EC00304=-798156,-183832
EC00305=-798156,-183832
EC00306=-798156,-183832
EC00307=-798156,-183832
EC00308=-798156,-183832
EC00309=-798156,-183832
EC00310=-798156,-183832
EC00311=-798156,-183832
EC00312=-798156,-183832
EC00313=-798156,-183832
EC00314=-798156,-183832
EC00315=-798156,-183832
EC00316=-798156,-183832
EC00317=-798156,-183832
EC00318=-798156,-183832
EC00319=-798156,-183832
EC00320=-798156,-183832
EC00321=-798156,-183832
EC00322=-798156,-183832
EC00323=-798156,-183832
EC00324=-798156,-183832
EC00325=-798156,-183832
EC00326=-798156,-183832
EC00327=-798156,-183832
EC00328=-798156,-183832
EC00329=-798156,-183832
EC00330=-798156,-183832
EC00331=-798156,-183832
EC00332=-798156,-183832
EC00333=-798156,-183832
EC00334=-798156,-183832
EC00335=-798156,-183832
EC00336=-798156,-183832
EC00337=-798156,-183832
EC00338=-798156,-183832
EC00339=-798156,-183832
EC00340=-798156,-183832
EC00341=-798156,-183832
EC00342=-798156,-183832
EC00343=-798156,-183832
EC00344=-798156,-183832
EC00345=-798156,-183832
EC00346=-798156,-183832
EC00347=-798156,-183832
EC00348=-798156,-183832
EC00349=-798156,-183832
EC00350=-798156,-183832
EC00351=-798156,-183832
EC00352=-798154,-183833
EC00353=-798156,-183832
EC00354=-798156,-183832
EC00355=-798156,-183832
EC00356=-798156,-183832
EC00357=-798156,-183832
EC00358=-798156,-183832
EC00359=-798156,-183832
EC00360=-798156,-183832
EC00361=-798156,-183832
EC00362=-798156,-183832
EC00363=-798156,-183832
EC00364=-798156,-183832
EC00365=-798156,-183832
EC00366=-798156,-183832
EC00367=-798156,-183832
EC00368=-798156,-183832
EC00369=-798156,-183832
EC00370=-798156,-183832
EC00371=-798156,-183832
EC00372=-798156,-183832
EC00373=-798156,-183832
EC00374=-798156,-183832
EC00375=-798156,-183832
EC00376=-798156,-183832
EC00377=-798156,-183832
EC00378=-798156,-183832
EC00379=-798156,-183832
EC00380=-798156,-183832
EC00381=-798156,-183832
EC00382=-798156,-183832
EC00383=-798156,-183832
EC00384=-798156,-183832
EC00385=-798156,-183832
EC00386=-798156,-183832
EC00387=-798156,-183832
EC00388=-798156,-183832
EC00389=-798156,-183832
EC00390=-798156,-183832
EC00391=-798156,-183832
EC00392=-798156,-183832
///POSTYPE BASE
///RECTAN
///RCONF 0,0,0,0,1,0,0,0,0,0,0,0,0,0,0,0,0,0,0,0,0,0,0,0
P00006=2.006,1.622,-0.565,0.0000,0.0000,0.0000
P00021=0.073,2.058,-0.109,0.0000,0.0000,0.0000
P00022=2.006,1.622,-0.565,0.0000,0.0000,0.0000
///RCONF 0,0,0,0,0,0,0,0,0,0,0,0,0,0,0,0,0,0,0,0,0,0,0,0
P00023=-2.957,-4.083,2.762,0.0000,0.0000,0.0000
P00031=-0.170,0.039,-0.647,0.0000,0.0000,0.0000
P00032=-0.423,0.157,3.222,0.0000,0.0000,0.0000
P00033=0.854,-1.099,3.047,0.0000,0.0000,0.0000
P00041=-0.109,0.014,0.966,0.0000,0.0000,0.0000
P00042=-0.220,0.371,-0.613,0.0000,0.0000,0.0000
P00043=-0.179,-5.890,-3.227,0.0000,0.0000,0.0000
P00051=-5.945,4.696,-10.293,0.0000,0.0000,0.0000
P00052=-0.153,5.586,-7.982,0.0000,0.0000,0.0000
P00053=0.015,-0.644,-4.942,0.0000,0.0000,0.0000
P00061=1211.499,975.999,-261.374,0.5148,35.2356,175.5099
P00062=1205.574,689.500,-262.704,0.5159,35.2461,175.5270
P00063=1197.217,207.358,-268.729,0.4863,35.2395,175.4586
//INST
///DATE 2024/12/17 12:40
///ATTR SC,RW
///GROUP1 RB1,BS1
///GROUP2 ST1
NOP
'X2_55b(90,0)
'
MOVJ C00000 BC00000 VJ=100.00  +MOVJ EC00000 VJ=100.00
MOVJ C00001 BC00001 VJ=100.00  +MOVJ EC00001 VJ=100.00
'Path S4425
SFTOF3D
MOVJ C00002 BC00002 VJ=100.00  +MOVJ EC00002 VJ=100.00
MOVL C00003 BC00003 V=800.0  +MOVJ EC00003 VJ=100.00
SMOVL C00004 BC00004 V=166.7  +MOVJ EC00004
SREFP 3 C00005 BC00005  +REFP EC00005
CALL JOB:SEARCH-R1-S13D
SET P021 P006
SFTON3D P021
SMOVL C00006 BC00006 V=166.7  +MOVJ EC00006
SMOVL C00007 BC00007 V=166.7  +MOVJ EC00007
SREFP 3 C00008 BC00008  +REFP EC00008
CALL JOB:SEARCH-R1-S13D
SET P021 P006
SFTON3D P021
SMOVL C00009 BC00009 V=166.7  +MOVJ EC00009
SMOVL C00010 BC00010 V=166.7  +MOVJ EC00010
SREFP 3 C00011 BC00011  +REFP EC00011
CALL JOB:SEARCH-R1-S13D
SET P021 P006
SFTON3D P021
SMOVL C00012 BC00012 V=166.7  +MOVJ EC00012
MOVL C00013 BC00013 V=800.0  +MOVJ EC00013 VJ=100.00
MOVL C00014 BC00014 V=1000.0  +MOVJ EC00014 VJ=100.00
'EndPath S4425
'Path S4426
SFTOF3D
MOVJ C00015 BC00015 VJ=100.00  +MOVJ EC00015 VJ=100.00
MOVL C00016 BC00016 V=800.0  +MOVJ EC00016 VJ=100.00
SMOVL C00017 BC00017 V=166.7  +MOVJ EC00017
SREFP 3 C00018 BC00018  +REFP EC00018
CALL JOB:SEARCH-R1-S13D
SET P022 P006
SFTON3D P022
SMOVL C00019 BC00019 V=166.7  +MOVJ EC00019
SMOVL C00020 BC00020 V=166.7  +MOVJ EC00020
SREFP 3 C00021 BC00021  +REFP EC00021
CALL JOB:SEARCH-R1-S13D
SET P022 P006
SFTON3D P022
SMOVL C00022 BC00022 V=166.7  +MOVJ EC00022
MOVL C00023 BC00023 V=800.0  +MOVJ EC00023 VJ=100.00
MOVL C00024 BC00024 V=1000.0  +MOVJ EC00024 VJ=100.00
'EndPath S4426
MOVJ C00025 BC00025 VJ=100.00  +MOVJ EC00025 VJ=100.00
'
MOVJ C00026 BC00026 VJ=100.00  +MOVJ EC00026 VJ=100.00
'Path S4427
SFTOF3D
MOVJ C00027 BC00027 VJ=100.00  +MOVJ EC00027 VJ=100.00
MOVL C00028 BC00028 V=800.0  +MOVJ EC00028 VJ=100.00
SMOVL C00029 BC00029 V=166.7  +MOVJ EC00029
SREFP 3 C00030 BC00030  +REFP EC00030
CALL JOB:SEARCH-R1-S13D
SET P031 P006
SFTON3D P031
SMOVL C00031 BC00031 V=166.7  +MOVJ EC00031
SMOVL C00032 BC00032 V=166.7  +MOVJ EC00032
SREFP 3 C00033 BC00033  +REFP EC00033
CALL JOB:SEARCH-R1-S13D
SET P031 P006
SFTON3D P031
SMOVL C00034 BC00034 V=166.7  +MOVJ EC00034
SMOVL C00035 BC00035 V=166.7  +MOVJ EC00035
SREFP 3 C00036 BC00036  +REFP EC00036
CALL JOB:SEARCH-R1-S13D
SET P031 P006
SFTON3D P031
SMOVL C00037 BC00037 V=166.7  +MOVJ EC00037
MOVL C00038 BC00038 V=800.0  +MOVJ EC00038 VJ=100.00
MOVL C00039 BC00039 V=1000.0  +MOVJ EC00039 VJ=100.00
'EndPath S4427
'Path S4428
SFTOF3D
MOVJ C00040 BC00040 VJ=100.00  +MOVJ EC00040 VJ=100.00
MOVL C00041 BC00041 V=800.0  +MOVJ EC00041 VJ=100.00
SMOVL C00042 BC00042 V=166.7  +MOVJ EC00042
SREFP 3 C00043 BC00043  +REFP EC00043
CALL JOB:SEARCH-R1-S13D
SET P032 P006
SFTON3D P032
SMOVL C00044 BC00044 V=166.7  +MOVJ EC00044
SMOVL C00045 BC00045 V=166.7  +MOVJ EC00045
SREFP 3 C00046 BC00046  +REFP EC00046
CALL JOB:SEARCH-R1-S13D
SET P032 P006
SFTON3D P032
SMOVL C00047 BC00047 V=166.7  +MOVJ EC00047
MOVL C00048 BC00048 V=800.0  +MOVJ EC00048 VJ=100.00
MOVL C00049 BC00049 V=1000.0  +MOVJ EC00049 VJ=100.00
'EndPath S4428
MOVJ C00050 BC00050 VJ=100.00  +MOVJ EC00050 VJ=100.00
'
MOVJ C00051 BC00051 VJ=100.00  +MOVJ EC00051 VJ=100.00
'Path S4429
SFTOF3D
MOVJ C00052 BC00052 VJ=100.00  +MOVJ EC00052 VJ=100.00
MOVL C00053 BC00053 V=800.0  +MOVJ EC00053 VJ=100.00
SMOVL C00054 BC00054 V=166.7  +MOVJ EC00054
SREFP 3 C00055 BC00055  +REFP EC00055
CALL JOB:SEARCH-R1-S13D
SET P041 P006
SFTON3D P041
SMOVL C00056 BC00056 V=166.7  +MOVJ EC00056
SMOVL C00057 BC00057 V=166.7  +MOVJ EC00057
SREFP 3 C00058 BC00058  +REFP EC00058
CALL JOB:SEARCH-R1-S13D
SET P041 P006
SFTON3D P041
SMOVL C00059 BC00059 V=166.7  +MOVJ EC00059
SMOVL C00060 BC00060 V=166.7  +MOVJ EC00060
SREFP 3 C00061 BC00061  +REFP EC00061
CALL JOB:SEARCH-R1-S13D
SET P041 P006
SFTON3D P041
SMOVL C00062 BC00062 V=166.7  +MOVJ EC00062
MOVL C00063 BC00063 V=800.0  +MOVJ EC00063 VJ=100.00
MOVL C00064 BC00064 V=1000.0  +MOVJ EC00064 VJ=100.00
'EndPath S4429
'Path S4430
SFTOF3D
MOVJ C00065 BC00065 VJ=100.00  +MOVJ EC00065 VJ=100.00
MOVL C00066 BC00066 V=800.0  +MOVJ EC00066 VJ=100.00
SMOVL C00067 BC00067 V=166.7  +MOVJ EC00067
SREFP 3 C00068 BC00068  +REFP EC00068
CALL JOB:SEARCH-R1-S13D
SET P042 P006
SFTON3D P042
SMOVL C00069 BC00069 V=166.7  +MOVJ EC00069
SMOVL C00070 BC00070 V=166.7  +MOVJ EC00070
SREFP 3 C00071 BC00071  +REFP EC00071
CALL JOB:SEARCH-R1-S13D
SET P042 P006
SFTON3D P042
SMOVL C00072 BC00072 V=166.7  +MOVJ EC00072
MOVL C00073 BC00073 V=800.0  +MOVJ EC00073 VJ=100.00
MOVL C00074 BC00074 V=1000.0  +MOVJ EC00074 VJ=100.00
'EndPath S4430
MOVJ C00075 BC00075 VJ=100.00  +MOVJ EC00075 VJ=100.00
'
MOVJ C00076 BC00076 VJ=100.00  +MOVJ EC00076 VJ=100.00
'Path S4431
SFTOF3D
MOVJ C00077 BC00077 VJ=100.00  +MOVJ EC00077 VJ=100.00
MOVL C00078 BC00078 V=800.0  +MOVJ EC00078 VJ=100.00
SMOVL C00079 BC00079 V=166.7  +MOVJ EC00079
SREFP 3 C00080 BC00080  +REFP EC00080
CALL JOB:SEARCH-R1-S13D
SET P051 P006
SFTON3D P051
SMOVL C00081 BC00081 V=166.7  +MOVJ EC00081
SMOVL C00082 BC00082 V=166.7  +MOVJ EC00082
SREFP 3 C00083 BC00083  +REFP EC00083
CALL JOB:SEARCH-R1-S13D
SET P051 P006
SFTON3D P051
SMOVL C00084 BC00084 V=166.7  +MOVJ EC00084
SMOVL C00085 BC00085 V=166.7  +MOVJ EC00085
SREFP 3 C00086 BC00086  +REFP EC00086
CALL JOB:SEARCH-R1-S13D
SET P051 P006
SFTON3D P051
SMOVL C00087 BC00087 V=250.0  +MOVJ EC00087
MOVL C00088 BC00088 V=1000.0  +MOVJ EC00088 VJ=100.00
'EndPath S4431
'Path S4432
SFTOF3D
MOVJ C00089 BC00089 VJ=100.00  +MOVJ EC00089 VJ=100.00
MOVL C00090 BC00090 V=800.0  +MOVJ EC00090 VJ=100.00
SMOVL C00091 BC00091 V=166.7  +MOVJ EC00091
SREFP 3 C00092 BC00092  +REFP EC00092
CALL JOB:SEARCH-R1-S13D
SET P052 P006
SFTON3D P052
SMOVL C00093 BC00093 V=166.7  +MOVJ EC00093
SMOVL C00094 BC00094 V=166.7  +MOVJ EC00094
SREFP 3 C00095 BC00095  +REFP EC00095
CALL JOB:SEARCH-R1-S13D
SET P052 P006
SFTON3D P052
SMOVL C00096 BC00096 V=166.7  +MOVJ EC00096
MOVL C00097 BC00097 V=800.0  +MOVJ EC00097 VJ=100.00
MOVL C00098 BC00098 V=1000.0  +MOVJ EC00098 VJ=100.00
'EndPath S4432
MOVJ C00099 BC00099 VJ=100.00  +MOVJ EC00099 VJ=100.00
'
MOVJ C00100 BC00100 VJ=100.00  +MOVJ EC00100 VJ=100.00
'Path S4433
SFTOF3D
MOVJ C00101 BC00101 VJ=100.00  +MOVJ EC00101 VJ=100.00
MOVL C00102 BC00102 V=800.0  +MOVJ EC00102 VJ=100.00
SMOVL C00103 BC00103 V=166.7  +MOVJ EC00103
SREFP 3 C00104 BC00104  +REFP EC00104
CALL JOB:SEARCH-R1-S13D
SET P061 P006
SFTON3D P061
SMOVL C00105 BC00105 V=166.7  +MOVJ EC00105
SMOVL C00106 BC00106 V=166.7  +MOVJ EC00106
SREFP 3 C00107 BC00107  +REFP EC00107
CALL JOB:SEARCH-R1-S13D
SET P061 P006
SFTON3D P061
SMOVL C00108 BC00108 V=166.7  +MOVJ EC00108
SMOVL C00109 BC00109 V=166.7  +MOVJ EC00109
SREFP 3 C00110 BC00110  +REFP EC00110
CALL JOB:SEARCH-R1-S13D
SET P061 P006
SFTON3D P061
SMOVL C00111 BC00111 V=166.7  +MOVJ EC00111
MOVL C00112 BC00112 V=800.0  +MOVJ EC00112 VJ=100.00
MOVL C00113 BC00113 V=1000.0  +MOVJ EC00113 VJ=100.00
'EndPath S4433
'Path S4434
SFTOF3D
MOVJ C00114 BC00114 VJ=100.00  +MOVJ EC00114 VJ=100.00
MOVL C00115 BC00115 V=800.0  +MOVJ EC00115 VJ=100.00
SMOVL C00116 BC00116 V=166.7  +MOVJ EC00116
SREFP 3 C00117 BC00117  +REFP EC00117
CALL JOB:SEARCH-R1-S13D
SET P062 P006
SFTON3D P062
SMOVL C00118 BC00118 V=166.7  +MOVJ EC00118
SMOVL C00119 BC00119 V=166.7  +MOVJ EC00119
SREFP 3 C00120 BC00120  +REFP EC00120
CALL JOB:SEARCH-R1-S13D
SET P062 P006
SFTON3D P062
SMOVL C00121 BC00121 V=166.7  +MOVJ EC00121
MOVL C00122 BC00122 V=800.0  +MOVJ EC00122 VJ=100.00
MOVL C00123 BC00123 V=1000.0  +MOVJ EC00123 VJ=100.00
'EndPath S4434
MOVJ C00124 BC00124 VJ=100.00  +MOVJ EC00124 VJ=100.00
MOVJ C00125 BC00125 VJ=100.00  +MOVJ EC00125 VJ=100.00
'
'Path S4435
SFTOF3D
MOVJ C00126 BC00126 VJ=100.00  +MOVJ EC00126 VJ=100.00
MOVL C00127 BC00127 V=800.0  +MOVJ EC00127 VJ=100.00
SMOVL C00128 BC00128 V=166.7  +MOVJ EC00128
SREFP 3 C00129 BC00129  +REFP EC00129
CALL JOB:SEARCH-R1-S13D
SET P063 P006
SFTON3D P063
SMOVL C00130 BC00130 V=166.7  +MOVJ EC00130
SMOVL C00131 BC00131 V=166.7  +MOVJ EC00131
SREFP 3 C00132 BC00132  +REFP EC00132
CALL JOB:SEARCH-R1-S13D
SET P063 P006
SFTON3D P063
SMOVL C00133 BC00133 V=166.7  +MOVJ EC00133
MOVL C00134 BC00134 V=800.0  +MOVJ EC00134 VJ=100.00
MOVL C00135 BC00135 V=1000.0  +MOVJ EC00135 VJ=100.00
'EndPath S4435
MOVJ C00136 BC00136 VJ=100.00  +MOVJ EC00136 VJ=100.00
MOVJ C00137 BC00137 VJ=100.00  +MOVJ EC00137 VJ=100.00
'Path S4436
SFTOF3D
MOVJ C00138 BC00138 VJ=100.00  +MOVJ EC00138 VJ=100.00
MOVL C00139 BC00139 V=800.0  +MOVJ EC00139 VJ=100.00
SMOVL C00140 BC00140 V=166.7  +MOVJ EC00140
SREFP 3 C00141 BC00141  +REFP EC00141
CALL JOB:SEARCH-R1-S13D
SET P053 P006
SFTON3D P053
SMOVL C00142 BC00142 V=166.7  +MOVJ EC00142
SMOVL C00143 BC00143 V=166.7  +MOVJ EC00143
SREFP 3 C00144 BC00144  +REFP EC00144
CALL JOB:SEARCH-R1-S13D
SET P053 P006
SFTON3D P053
SMOVL C00145 BC00145 V=166.7  +MOVJ EC00145
MOVL C00146 BC00146 V=800.0  +MOVJ EC00146 VJ=100.00
MOVL C00147 BC00147 V=1000.0  +MOVJ EC00147 VJ=100.00
'EndPath S4436
MOVJ C00148 BC00148 VJ=100.00  +MOVJ EC00148 VJ=100.00
MOVJ C00149 BC00149 VJ=100.00  +MOVJ EC00149 VJ=100.00
'Path S4437
SFTOF3D
MOVJ C00150 BC00150 VJ=100.00  +MOVJ EC00150 VJ=100.00
MOVL C00151 BC00151 V=800.0  +MOVJ EC00151 VJ=100.00
SMOVL C00152 BC00152 V=166.7  +MOVJ EC00152
SREFP 3 C00153 BC00153  +REFP EC00153
CALL JOB:SEARCH-R1-S13D
SET P043 P006
SFTON3D P043
SMOVL C00154 BC00154 V=166.7  +MOVJ EC00154
SREFP 3 C00155 BC00155  +REFP EC00155
CALL JOB:SEARCH-R1-S13D
SET P043 P006
SFTON3D P043
SMOVL C00156 BC00156 V=166.7  +MOVJ EC00156
MOVL C00157 BC00157 V=800.0  +MOVJ EC00157 VJ=100.00
MOVL C00158 BC00158 V=1000.0  +MOVJ EC00158 VJ=100.00
'EndPath S4437
MOVJ C00159 BC00159 VJ=100.00  +MOVJ EC00159 VJ=100.00
MOVJ C00160 BC00160 VJ=100.00  +MOVJ EC00160 VJ=100.00
'Path S4438
SFTOF3D
MOVJ C00161 BC00161 VJ=100.00  +MOVJ EC00161 VJ=100.00
MOVL C00162 BC00162 V=800.0  +MOVJ EC00162 VJ=100.00
SMOVL C00163 BC00163 V=166.7  +MOVJ EC00163
SREFP 3 C00164 BC00164  +REFP EC00164
CALL JOB:SEARCH-R1-S13D
SET P033 P006
SFTON3D P033
SMOVL C00165 BC00165 V=166.7  +MOVJ EC00165
SMOVL C00166 BC00166 V=166.7  +MOVJ EC00166
SREFP 3 C00167 BC00167  +REFP EC00167
CALL JOB:SEARCH-R1-S13D
SET P033 P006
SFTON3D P033
SMOVL C00168 BC00168 V=166.7  +MOVJ EC00168
MOVL C00169 BC00169 V=800.0  +MOVJ EC00169 VJ=100.00
MOVL C00170 BC00170 V=1000.0  +MOVJ EC00170 VJ=100.00
'EndPath S4438
MOVJ C00171 BC00171 VJ=100.00  +MOVJ EC00171 VJ=100.00
MOVJ C00172 BC00172 VJ=100.00  +MOVJ EC00172 VJ=100.00
'Path S4439
SFTOF3D
MOVJ C00173 BC00173 VJ=100.00  +MOVJ EC00173 VJ=100.00
MOVL C00174 BC00174 V=800.0  +MOVJ EC00174 VJ=100.00
SMOVL C00175 BC00175 V=166.7  +MOVJ EC00175
SREFP 3 C00176 BC00176  +REFP EC00176
CALL JOB:SEARCH-R1-S13D
SET P023 P006
SFTON3D P023
SMOVL C00177 BC00177 V=166.7  +MOVJ EC00177
SREFP 3 C00178 BC00178  +REFP EC00178
CALL JOB:SEARCH-R1-S13D
SET P023 P006
SFTON3D P023
SMOVL C00179 BC00179 V=166.7  +MOVJ EC00179
MOVL C00180 BC00180 V=800.0  +MOVJ EC00180 VJ=100.00
MOVL C00181 BC00181 V=1000.0  +MOVJ EC00181 VJ=100.00
'EndPath S4439
MOVJ C00182 BC00182 VJ=100.00  +MOVJ EC00182 VJ=100.00
'
'
'
MOVJ C00183 BC00183 VJ=100.00  +MOVJ EC00183 VJ=100.00
'Path W4440
SFTOF3D
SFTON3D P043
MOVJ C00184 BC00184 VJ=100.00  +MOVJ EC00184 VJ=100.00
SMOVL C00185 BC00185 V=800.0  +MOVJ EC00185
SMOVL C00186 BC00186 V=166.7 PL=0  +MOVJ EC00186
ARCON
SMOVL C00187 BC00187 V=10.0  +MOVJ EC00187
SMOVL C00188 BC00188 V=10.0  +MOVJ EC00188
SMOVL C00189 BC00189 V=10.0  +MOVJ EC00189
SMOVL C00190 BC00190 V=10.0  +MOVJ EC00190
SMOVL C00191 BC00191 V=10.0  +MOVJ EC00191
ARCOF
SMOVL C00192 BC00192 V=800.0  +MOVJ EC00192
SMOVL C00193 BC00193 V=1000.0  +MOVJ EC00193
SFTOF3D
'EndPath W4440
MOVJ C00194 BC00194 VJ=100.00  +MOVJ EC00194 VJ=100.00
MOVJ C00195 BC00195 VJ=100.00  +MOVJ EC00195 VJ=100.00
'Path W4441
SFTOF3D
SFTON3D P023
MOVJ C00196 BC00196 VJ=100.00  +MOVJ EC00196 VJ=100.00
SMOVL C00197 BC00197 V=800.0  +MOVJ EC00197
SMOVL C00198 BC00198 V=166.7 PL=0  +MOVJ EC00198
ARCON
SMOVL C00199 BC00199 V=10.0  +MOVJ EC00199
SMOVL C00200 BC00200 V=10.0  +MOVJ EC00200
SMOVL C00201 BC00201 V=10.0  +MOVJ EC00201
SMOVL C00202 BC00202 V=10.0  +MOVJ EC00202
ARCOF
SMOVL C00203 BC00203 V=800.0  +MOVJ EC00203
SMOVL C00204 BC00204 V=1000.0  +MOVJ EC00204
SFTOF3D
'EndPath W4441
MOVJ C00205 BC00205 VJ=100.00  +MOVJ EC00205 VJ=100.00
MOVJ C00206 BC00206 VJ=100.00  +MOVJ EC00206 VJ=100.00
'Path W4442
SFTOF3D
SFTON3D P063
MOVJ C00207 BC00207 VJ=100.00  +MOVJ EC00207 VJ=100.00
SMOVL C00208 BC00208 V=800.0  +MOVJ EC00208
SMOVL C00209 BC00209 V=166.7 PL=0  +MOVJ EC00209
ARCON
SMOVL C00210 BC00210 V=10.0  +MOVJ EC00210
SMOVL C00211 BC00211 V=10.0  +MOVJ EC00211
SMOVL C00212 BC00212 V=10.0  +MOVJ EC00212
SMOVL C00213 BC00213 V=10.0  +MOVJ EC00213
SMOVL C00214 BC00214 V=10.0  +MOVJ EC00214
SMOVL C00215 BC00215 V=10.0  +MOVJ EC00215
SMOVL C00216 BC00216 V=10.0  +MOVJ EC00216
SMOVL C00217 BC00217 V=10.0  +MOVJ EC00217
ARCOF
SMOVL C00218 BC00218 V=800.0  +MOVJ EC00218
SMOVL C00219 BC00219 V=1000.0  +MOVJ EC00219
SFTOF3D
'EndPath W4442
MOVJ C00220 BC00220 VJ=100.00  +MOVJ EC00220 VJ=100.00
MOVJ C00221 BC00221 VJ=100.00  +MOVJ EC00221 VJ=100.00
'Path W4443
SFTOF3D
SFTON3D P033
MOVJ C00222 BC00222 VJ=100.00  +MOVJ EC00222 VJ=100.00
SMOVL C00223 BC00223 V=800.0  +MOVJ EC00223
SMOVL C00224 BC00224 V=166.7 PL=0  +MOVJ EC00224
ARCON
SMOVL C00225 BC00225 V=10.0  +MOVJ EC00225
SMOVL C00226 BC00226 V=10.0  +MOVJ EC00226
SMOVL C00227 BC00227 V=10.0  +MOVJ EC00227
SMOVL C00228 BC00228 V=10.0  +MOVJ EC00228
SMOVL C00229 BC00229 V=10.0  +MOVJ EC00229
SMOVL C00230 BC00230 V=10.0  +MOVJ EC00230
SMOVL C00231 BC00231 V=10.0  +MOVJ EC00231
SMOVL C00232 BC00232 V=10.0  +MOVJ EC00232
ARCOF
SMOVL C00233 BC00233 V=800.0  +MOVJ EC00233
SMOVL C00234 BC00234 V=1000.0  +MOVJ EC00234
SFTOF3D
'EndPath W4443
MOVJ C00235 BC00235 VJ=100.00  +MOVJ EC00235 VJ=100.00
MOVJ C00236 BC00236 VJ=100.00  +MOVJ EC00236 VJ=100.00
'Path W4444
SFTOF3D
SFTON3D P053
MOVJ C00237 BC00237 VJ=100.00  +MOVJ EC00237 VJ=100.00
SMOVL C00238 BC00238 V=800.0  +MOVJ EC00238
SMOVL C00239 BC00239 V=166.7 PL=0  +MOVJ EC00239
ARCON
SMOVL C00240 BC00240 V=10.0  +MOVJ EC00240
SMOVL C00241 BC00241 V=10.0  +MOVJ EC00241
SMOVL C00242 BC00242 V=10.0  +MOVJ EC00242
SMOVL C00243 BC00243 V=10.0  +MOVJ EC00243
SMOVL C00244 BC00244 V=10.0  +MOVJ EC00244
SMOVL C00245 BC00245 V=10.0  +MOVJ EC00245
SMOVL C00246 BC00246 V=10.0  +MOVJ EC00246
ARCOF
SMOVL C00247 BC00247 V=800.0  +MOVJ EC00247
SMOVL C00248 BC00248 V=1000.0  +MOVJ EC00248
SFTOF3D
'EndPath W4444
MOVJ C00249 BC00249 VJ=100.00  +MOVJ EC00249 VJ=100.00
'
MOVJ C00250 BC00250 VJ=100.00  +MOVJ EC00250 VJ=100.00
MOVJ C00251 BC00251 VJ=100.00  +MOVJ EC00251 VJ=100.00
'Path W4445
SFTOF3D
SFTON3D P042
MOVJ C00252 BC00252 VJ=100.00  +MOVJ EC00252 VJ=100.00
SMOVL C00253 BC00253 V=800.0  +MOVJ EC00253
SMOVL C00254 BC00254 V=166.7 PL=0  +MOVJ EC00254
ARCON
SMOVL C00255 BC00255 V=10.0  +MOVJ EC00255
SMOVL C00256 BC00256 V=10.0  +MOVJ EC00256
SMOVL C00257 BC00257 V=10.0  +MOVJ EC00257
SMOVL C00258 BC00258 V=10.0  +MOVJ EC00258
ARCOF
SMOVL C00259 BC00259 V=800.0  +MOVJ EC00259
SMOVL C00260 BC00260 V=1000.0  +MOVJ EC00260
SFTOF3D
'EndPath W4445
'Path W4446
SFTOF3D
SFTON3D P041
MOVJ C00261 BC00261 VJ=100.00  +MOVJ EC00261 VJ=100.00
SMOVL C00262 BC00262 V=800.0  +MOVJ EC00262
SMOVL C00263 BC00263 V=166.7 PL=0  +MOVJ EC00263
ARCON
SMOVL C00264 BC00264 V=10.0  +MOVJ EC00264
SMOVL C00265 BC00265 V=10.0  +MOVJ EC00265
SMOVL C00266 BC00266 V=10.0  +MOVJ EC00266
SMOVL C00267 BC00267 V=10.0  +MOVJ EC00267
ARCOF
SMOVL C00268 BC00268 V=800.0  +MOVJ EC00268
SMOVL C00269 BC00269 V=1000.0  +MOVJ EC00269
SFTOF3D
'EndPath W4446
'Path W4447
SFTOF3D
SFTON3D P041
MOVJ C00270 BC00270 VJ=100.00  +MOVJ EC00270 VJ=100.00
SMOVL C00271 BC00271 V=800.0  +MOVJ EC00271
SMOVL C00272 BC00272 V=166.7 PL=0  +MOVJ EC00272
ARCON
SMOVL C00273 BC00273 V=10.0  +MOVJ EC00273
SMOVL C00274 BC00274 V=10.0  +MOVJ EC00274
SMOVL C00275 BC00275 V=10.0  +MOVJ EC00275
ARCOF
SMOVL C00276 BC00276 V=800.0  +MOVJ EC00276
SMOVL C00277 BC00277 V=1000.0  +MOVJ EC00277
SFTOF3D
'EndPath W4447
MOVJ C00278 BC00278 VJ=100.00  +MOVJ EC00278 VJ=100.00
'
'
MOVJ C00279 BC00279 VJ=100.00  +MOVJ EC00279 VJ=100.00
'Path W4448
SFTOF3D
SFTON3D P022
MOVJ C00280 BC00280 VJ=100.00  +MOVJ EC00280 VJ=100.00
SMOVL C00281 BC00281 V=800.0  +MOVJ EC00281
SMOVL C00282 BC00282 V=166.7 PL=0  +MOVJ EC00282
MACRO1 MJ#(0) ARGF9
ARCON
SMOVL C00283 BC00283 V=10.0  +MOVJ EC00283
SMOVL C00284 BC00284 V=10.0  +MOVJ EC00284
SMOVL C00285 BC00285 V=10.0  +MOVJ EC00285
SMOVL C00286 BC00286 V=10.0  +MOVJ EC00286
SMOVL C00287 BC00287 V=10.0  +MOVJ EC00287
ARCOF
SMOVL C00288 BC00288 V=800.0  +MOVJ EC00288
SMOVL C00289 BC00289 V=1000.0  +MOVJ EC00289
SFTOF3D
'EndPath W4448
'Path W4449
SFTOF3D
SFTON3D P021
MOVJ C00290 BC00290 VJ=100.00  +MOVJ EC00290 VJ=100.00
SMOVL C00291 BC00291 V=800.0  +MOVJ EC00291
SMOVL C00292 BC00292 V=166.7 PL=0  +MOVJ EC00292
ARCON
SMOVL C00293 BC00293 V=10.0  +MOVJ EC00293
SMOVL C00294 BC00294 V=10.0  +MOVJ EC00294
SMOVL C00295 BC00295 V=10.0  +MOVJ EC00295
SMOVL C00296 BC00296 V=10.0  +MOVJ EC00296
SMOVL C00297 BC00297 V=10.0  +MOVJ EC00297
ARCOF
SMOVL C00298 BC00298 V=800.0  +MOVJ EC00298
SMOVL C00299 BC00299 V=1000.0  +MOVJ EC00299
SFTOF3D
'EndPath W4449
'Path W4450
SFTOF3D
SFTON3D P021
MOVJ C00300 BC00300 VJ=100.00  +MOVJ EC00300 VJ=100.00
SMOVL C00301 BC00301 V=800.0  +MOVJ EC00301
SMOVL C00302 BC00302 V=166.7 PL=0  +MOVJ EC00302
ARCON
SMOVL C00303 BC00303 V=10.0  +MOVJ EC00303
SMOVL C00304 BC00304 V=10.0  +MOVJ EC00304
SMOVL C00305 BC00305 V=10.0  +MOVJ EC00305
ARCOF
SMOVL C00306 BC00306 V=800.0  +MOVJ EC00306
SMOVL C00307 BC00307 V=1000.0  +MOVJ EC00307
SFTOF3D
'EndPath W4450
MOVJ C00308 BC00308 VJ=100.00  +MOVJ EC00308 VJ=100.00
'
'
MOVJ C00309 BC00309 VJ=100.00  +MOVJ EC00309 VJ=100.00
'Path W4451
SFTOF3D
SFTON3D P062
MOVJ C00310 BC00310 VJ=100.00  +MOVJ EC00310 VJ=100.00
SMOVL C00311 BC00311 V=800.0  +MOVJ EC00311
SMOVL C00312 BC00312 V=166.7 PL=0  +MOVJ EC00312
ARCON
SMOVL C00313 BC00313 V=10.0  +MOVJ EC00313
SMOVL C00314 BC00314 V=10.0  +MOVJ EC00314
SMOVL C00315 BC00315 V=10.0  +MOVJ EC00315
ARCOF
SMOVL C00316 BC00316 V=800.0  +MOVJ EC00316
SMOVL C00317 BC00317 V=1000.0  +MOVJ EC00317
SFTOF3D
'EndPath W4451
'Path W4452
SFTOF3D
SFTON3D P061
MOVJ C00318 BC00318 VJ=100.00  +MOVJ EC00318 VJ=100.00
MACRO1 MJ#(0) ARGF21
SMOVL C00319 BC00319 V=800.0  +MOVJ EC00319
SMOVL C00320 BC00320 V=166.7 PL=0  +MOVJ EC00320
ARCON
SMOVL C00321 BC00321 V=10.0  +MOVJ EC00321
SMOVL C00322 BC00322 V=10.0  +MOVJ EC00322
SMOVL C00323 BC00323 V=10.0  +MOVJ EC00323
SMOVL C00324 BC00324 V=10.0  +MOVJ EC00324
ARCOF
SMOVL C00325 BC00325 V=800.0  +MOVJ EC00325
SMOVL C00326 BC00326 V=1000.0  +MOVJ EC00326
SFTOF3D
'EndPath W4452
'Path W4453
SFTOF3D
SFTON3D P061
MOVJ C00327 BC00327 VJ=100.00  +MOVJ EC00327 VJ=100.00
SMOVL C00328 BC00328 V=800.0  +MOVJ EC00328
SMOVL C00329 BC00329 V=166.7 PL=0  +MOVJ EC00329
ARCON
SMOVL C00330 BC00330 V=10.0  +MOVJ EC00330
SMOVL C00331 BC00331 V=10.0  +MOVJ EC00331
SMOVL C00332 BC00332 V=10.0  +MOVJ EC00332
ARCOF
SMOVL C00333 BC00333 V=800.0  +MOVJ EC00333
SMOVL C00334 BC00334 V=1000.0  +MOVJ EC00334
SFTOF3D
'EndPath W4453
MOVJ C00335 BC00335 VJ=100.00  +MOVJ EC00335 VJ=100.00
'
'
MOVJ C00336 BC00336 VJ=100.00  +MOVJ EC00336 VJ=100.00
'Path W4454
SFTOF3D
SFTON3D P032
MOVJ C00337 BC00337 VJ=100.00  +MOVJ EC00337 VJ=100.00
SMOVL C00338 BC00338 V=800.0  +MOVJ EC00338
SMOVL C00339 BC00339 V=166.7 PL=0  +MOVJ EC00339
ARCON
SMOVL C00340 BC00340 V=10.0  +MOVJ EC00340
SMOVL C00341 BC00341 V=10.0  +MOVJ EC00341
SMOVL C00342 BC00342 V=10.0  +MOVJ EC00342
SMOVL C00343 BC00343 V=10.0  +MOVJ EC00343
ARCOF
SMOVL C00344 BC00344 V=800.0  +MOVJ EC00344
SMOVL C00345 BC00345 V=1000.0  +MOVJ EC00345
SFTOF3D
'EndPath W4454
'Path W4455
SFTOF3D
SFTON3D P031
MOVJ C00346 BC00346 VJ=100.00  +MOVJ EC00346 VJ=100.00
SMOVL C00347 BC00347 V=800.0  +MOVJ EC00347
SMOVL C00348 BC00348 V=166.7 PL=0  +MOVJ EC00348
ARCON
SMOVL C00349 BC00349 V=10.0  +MOVJ EC00349
SMOVL C00350 BC00350 V=10.0  +MOVJ EC00350
SMOVL C00351 BC00351 V=10.0  +MOVJ EC00351
SMOVL C00352 BC00352 V=10.0  +MOVJ EC00352
ARCOF
SMOVL C00353 BC00353 V=800.0  +MOVJ EC00353
SMOVL C00354 BC00354 V=1000.0  +MOVJ EC00354
SFTOF3D
'EndPath W4455
'Path W4456
SFTOF3D
SFTON3D P031
MOVJ C00355 BC00355 VJ=100.00  +MOVJ EC00355 VJ=100.00
SMOVL C00356 BC00356 V=800.0  +MOVJ EC00356
SMOVL C00357 BC00357 V=166.7 PL=0  +MOVJ EC00357
ARCON
SMOVL C00358 BC00358 V=10.0  +MOVJ EC00358
SMOVL C00359 BC00359 V=10.0  +MOVJ EC00359
SMOVL C00360 BC00360 V=10.0  +MOVJ EC00360
ARCOF
SMOVL C00361 BC00361 V=800.0  +MOVJ EC00361
SMOVL C00362 BC00362 V=1000.0  +MOVJ EC00362
SFTOF3D
'EndPath W4456
MOVJ C00363 BC00363 VJ=100.00  +MOVJ EC00363 VJ=100.00
'
'
MOVJ C00364 BC00364 VJ=100.00  +MOVJ EC00364 VJ=100.00
'Path W4457
SFTOF3D
SFTON3D P052
MOVJ C00365 BC00365 VJ=100.00  +MOVJ EC00365 VJ=100.00
SMOVL C00366 BC00366 V=800.0  +MOVJ EC00366
MACRO1 MJ#(0) ARGF14
SMOVL C00367 BC00367 V=166.7 PL=0  +MOVJ EC00367
ARCON
SMOVL C00368 BC00368 V=10.0  +MOVJ EC00368
SMOVL C00369 BC00369 V=10.0  +MOVJ EC00369
SMOVL C00370 BC00370 V=10.0  +MOVJ EC00370
SMOVL C00371 BC00371 V=10.0  +MOVJ EC00371
ARCOF
SMOVL C00372 BC00372 V=800.0  +MOVJ EC00372
SMOVL C00373 BC00373 V=1000.0  +MOVJ EC00373
SFTOF3D
'EndPath W4457
'Path W4458
SFTOF3D
SFTON3D P051
MOVJ C00374 BC00374 VJ=100.00  +MOVJ EC00374 VJ=100.00
SMOVL C00375 BC00375 V=800.0  +MOVJ EC00375
MACRO1 MJ#(0) ARGF21
SMOVL C00376 BC00376 V=166.7 PL=0  +MOVJ EC00376
ARCON
SMOVL C00377 BC00377 V=10.0  +MOVJ EC00377
SMOVL C00378 BC00378 V=10.0  +MOVJ EC00378
SMOVL C00379 BC00379 V=10.0  +MOVJ EC00379
SMOVL C00380 BC00380 V=10.0  +MOVJ EC00380
ARCOF
SMOVL C00381 BC00381 V=800.0  +MOVJ EC00381
SMOVL C00382 BC00382 V=1000.0  +MOVJ EC00382
SFTOF3D
'EndPath W4458
'Path W4459
SFTOF3D
SFTON3D P051
MOVJ C00383 BC00383 VJ=100.00  +MOVJ EC00383 VJ=100.00
SMOVL C00384 BC00384 V=800.0  +MOVJ EC00384
SMOVL C00385 BC00385 V=166.7 PL=0  +MOVJ EC00385
ARCON
SMOVL C00386 BC00386 V=10.0  +MOVJ EC00386
SMOVL C00387 BC00387 V=10.0  +MOVJ EC00387
SMOVL C00388 BC00388 V=10.0  +MOVJ EC00388
ARCOF
SMOVL C00389 BC00389 V=800.0  +MOVJ EC00389
SMOVL C00390 BC00390 V=1000.0  +MOVJ EC00390
SFTOF3D
'EndPath W4459
MOVJ C00391 BC00391 VJ=100.00  +MOVJ EC00391 VJ=100.00
MOVJ C00392 BC00392 VJ=100.00  +MOVJ EC00392 VJ=100.00
'
END
